{attribute 'GeneratedUsingTerminal: EL7031-0030-0016'}
{attribute addProperty BoxType "EL7031-0030-0016"}
{attribute addProperty Id "EtcSlaveTerminalBaseENC_Status_compactAT %I*ENC_Status_compact_3C6E2C4411STM_StatusAT %I*STM_Status_36ED096F11AI_Standard_Channel_1AT %I*AI_Standard_Channel_205D8A067AI_Standard_Channel_2AT %I*AI_Standard_Channel_205D8A067ENC_Control_compactAT %Q*ENC_Control_compact_2E82BC435STM_ControlAT %Q*STM_Control_5A8B50163STM_VelocityAT %Q*STM_Velocity_A47A3F412WcStateAT %I*WcState_9091E0EB2InfoDataAT %I*InfoData_939F71B614"}
{attribute addProperty CRC "946338507"}
{attribute addProperty Size "62"}
TYPE EL7031_3867FACB EXTENDS EtcSlaveTerminalBase :
STRUCT
	{attribute addProperty Name "ENC_Status_compact"}
	ENC_Status_compact : ENC_Status_compact_3C6E2C44;
	{attribute addProperty Name "STM_Status"}
	STM_Status : STM_Status_36ED096F;
	{attribute addProperty Name "AI_Standard_Channel_1"}
	AI_Standard_Channel_1 : AI_Standard_Channel_205D8A06;
	{attribute addProperty Name "AI_Standard_Channel_2"}
	AI_Standard_Channel_2 : AI_Standard_Channel_205D8A06;
	{attribute addProperty Name "ENC_Control_compact"}
	ENC_Control_compact : ENC_Control_compact_2E82BC43;
	{attribute addProperty Name "STM_Control"}
	STM_Control : STM_Control_5A8B5016;
	{attribute addProperty Name "STM_Velocity"}
	STM_Velocity : STM_Velocity_A47A3F41;
	{attribute addProperty Name "WcState"}
	WcState : WcState_9091E0EB;
	{attribute addProperty Name "InfoData"}
	InfoData : InfoData_939F71B6;
END_STRUCT
END_TYPE

(* stored: Version 1.2.0.0, ProductVersion 3.1.4024.9
   DUT EL7031_3867FACB: Id {350af9fe-2d78-48d9-a5c2-8db3df0e9510} *)
